// TIA Portal V20 export
TYPE "LER_TypeFATMode_ModeSelect"
// stored: Access Published
   STRUCT
      HoursTestMode : Bool;
      CapabilityMode : Bool;
      SamplingMode : Bool;
   END_STRUCT;
END_TYPE
